KUKA KRL program: chk_w3_grp5_clo.src

&ACCESS RVO1
&COMMENT Check GRP Z5 ACTROS CLOSE
DEF chk_w3_grp5_clo( )

; Check gripper actros CLOSE Z5
;//---- Start User-------

$TIMER[10] = 0
$TIMER_STOP[10] = FALSE

WAIT FOR ($IN[28])
WAIT FOR (NOT $IN[27])

$TIMER_STOP[10] = TRUE
$TIMER[10] = 0

;//---- End User---------

END
